FUNCTION_BLOCK WStrMem
VAR_INPUT
END_VAR
VAR_OUTPUT
END_VAR
VAR
	mem : WSTRING;
END_VAR

METHOD APPEND : BOOL
VAR_INPUT
	STR : WSTRING;
END_VAR
mem := WCONCAT(mem , STR);
END_METHOD

METHOD INSERT : BOOL
VAR_INPUT
	STR : WSTRING;
END_VAR
mem := WCONCAT(STR, mem);
END_METHOD

PROPERTY READ : WSTRING
GET
READ := mem;
END_GET
END_PROPERTY

METHOD WRITE : BOOL
VAR_INPUT
	STR :WSTRING;
END_VAR
mem := STR;
END_METHOD

END_FUNCTION_BLOCK

(* stored: Version 1.1.0.1, ProductVersion 3.1.4026.13
   POU WStrMem: Id {4bc9294e-cf92-4dcc-8c1c-8bf714633a81}, SpecialFunc None
   Method APPEND: Id {eafada67-54c0-4ea0-8c0d-7041761f58eb}
   Method INSERT: Id {8874ca3e-c338-4eeb-aa0f-67310d15cb16}
   Property READ: Id {bacf7e6b-e71b-4cd9-bd46-50fbc427eb00}
   Get Get: Id {69b2fdd1-cef1-4488-8810-e75e8ee6de57}
   Method WRITE: Id {a2974a77-ebeb-45f1-8bbc-8a4b44e731dc} *)
